VAR_GLOBAL
END_VAR

(* stored: Version 1.1.0.1, ProductVersion 3.1.0.19
   GVL MER_CmdState: Id {b9214a5f-7159-4b63-935d-ec28da4fcc76} *)
